Staubli VAL3: Control_Para1.pgx

public program Control_Para1(trsf& x_trTrsf, bool& x_bRes, bool x_bCut, num x_nType)
  local string l_sItem[6]
  local num l_nNum
  local num l_nKey
  local num l_nData[6]
  local num l_nSelectIndex
begin
  //为LasMAN3.7进行配置
  //修改点位的参数


  //通过局部变量来实现内部存储
  l_nData[3]=x_trTrsf.x
  l_nData[4]=x_trTrsf.y
  l_nData[0]=x_trTrsf.z
  l_nData[1]=x_trTrsf.rx

  l_nData[2]=x_trTrsf.ry
  l_nData[5]=x_trTrsf.rz
  l_nNum=sel(x_bRes,1,0)

  //界面初始化
  resize(sData,1,2)
  if x_bCut

    sData[0]="直线"
    sData[1]="圆弧"
    l_sItem[0]="速度(mm/s:"+toString(".3",l_nData[0])
    l_sItem[1]="加速度(%):"+toString(".3",l_nData[1])
    l_sItem[2]="BLend(mm):"+toString(".3",l_nData[2])
    l_sItem[3]="工艺     :"+toString(".3",l_nData[3])
    l_sItem[4]="动作     :"+toString(".3",l_nData[4])
    l_sItem[5]="圆弧/直线:"+sData[l_nNum]

  else
    sData[0]="MoveJ"
    sData[1]="MoveL"
    l_sItem[0]="速度(mm/s:"+toString(".3",l_nData[0])
    l_sItem[1]="加速度(%):"+toString(".3",l_nData[1])
    l_sItem[2]="关节/直线:"+sData[l_nNum]

  endIf

  call Control_BottomS(",,,,,,取消,确定")
  if x_bCut
    if x_nType!=10
      call Control_PanelXY(8,0,18,5)
    else
      call Control_PanelXY(8,0,18,6)
    endIf
  else
    call Control_PanelXY(8,0,17,3)
  endIf
  call Control_Panel("参数")
  call Control_List(l_sItem,l_nSelectIndex)


  //按键响应
  while true
    l_nKey=getKey()

    switch l_nKey
      case 261
        l_nSelectIndex=max(0,l_nSelectIndex-1)
      break

      case 266
        if x_bCut
          if x_nType==10
            l_nSelectIndex=min(l_nSelectIndex+1,5)
          else
            l_nSelectIndex=min(l_nSelectIndex+1,4)
          endIf
        else
          l_nSelectIndex=min(l_nSelectIndex+1,2)
        endIf
      break

      case 278
        x_trTrsf.x=l_nData[3]
        x_trTrsf.y=l_nData[4]
        x_trTrsf.z=l_nData[0]
        x_trTrsf.rx=l_nData[1]

        x_trTrsf.ry=l_nData[2]
        x_trTrsf.rz=l_nData[5]
        x_bRes=(l_nNum==1)
        cls()
        return
      break


      case 277,255
        cls()
        return
      break



      case 270
        if (l_nSelectIndex==2 and !x_bCut) or (l_nSelectIndex==5 and x_bCut)
          call Sel_Edit(l_nNum,nPanelLTopX+11,l_nSelectIndex+nPanelLTopY+1,sData)

        else
          call Float_Edit(l_nData[l_nSelectIndex],nPanelLTopX+11,l_nSelectIndex+nPanelLTopY+1)
        endIf
      break

    endSwitch

    if l_nKey!=-1
      if x_bCut

        sData[0]="直线"
        sData[1]="圆弧"
        l_sItem[0]="速度(mm/s:"+toString(".3",l_nData[0])
        l_sItem[1]="加速度(%):"+toString(".3",l_nData[1])
        l_sItem[2]="BLend(mm):"+toString(".3",l_nData[2])
        l_sItem[3]="工艺     :"+toString(".3",l_nData[3])
        l_sItem[4]="动作     :"+toString(".3",l_nData[4])
        l_sItem[5]="圆弧/直线:"+sData[l_nNum]

      else
        sData[0]="MoveJ"
        sData[1]="MoveL"
        l_sItem[0]="速度(mm/s:"+toString(".3",l_nData[0])
        l_sItem[1]="加速度(%):"+toString(".3",l_nData[1])
        l_sItem[2]="关节/直线:"+sData[l_nNum]

      endIf
      call Control_List(l_sItem,l_nSelectIndex)

    endIf






  endWhile

end
